FUNCTION_BLOCK FB_SaMElementProduction EXTENDS FB_SaMElement
VAR
END_VAR

END_FUNCTION_BLOCK

(* stored: Version 1.1.0.1
   POU FB_SaMElementProduction: Id {2553c4ee-ccbe-09f4-23d8-9032ffb84f10}, SpecialFunc None *)
